PROGRAM INTERNAL PRG_TEST_FB_PARFILEHANDLER
VAR
	bEnableTests : BOOL;
	fbParFileHandler: FB_ParameterFileHandler;
	stParameter 	: Udt_Parameter; // NOTE: Udt_Parameter is persistent
	bAddParameter 	: BOOL;
	bInit			: BOOL;
	bCmdSavePar		: BOOL;
END_VAR

IF bEnableTests THEN
	fbParFileHandler();
	
	IF bAddParameter THEN
		bAddParameter := FALSE;
		fbParFileHandler.CmdAddParameter(stParameter);
	END_IF
	
	IF bInit THEN
		bInit R= fbParFileHandler.Init();
	END_IF
	
	IF bCmdSavePar THEN
		bCmdSavePar R= fbParFileHandler.CmdSavePar();
	END_IF
END_IF

END_PROGRAM

(* stored: Version 1.1.0.1, ProductVersion 3.1.4024.11
   POU PRG_TEST_FB_PARFILEHANDLER: Id {9f293204-c2aa-0fe1-1474-f57aeffff999}, SpecialFunc None *)
